Fanuc KAREL source: IN_RANGE.kl

PROGRAM T
%NOLOCKGROUP
VAR
 v0 : XYZWPREXT
 res : BOOLEAN
BEGIN
 res = IN_RANGE(v0)
END T
